LIN {X 0,Y 131.799,Z 543.633,A -85,B 0,C 180,E1 -35494.427,E2 -35494.427} C_VEL
LIN {X 0,Y 126.443,Z 556.276,A -85,B 0,C 180,E1 -35496.559,E2 -35496.559} C_VEL
LIN {X 0,Y 120.613,Z 567.576,A -85,B 0,C 180,E1 -35499.038,E2 -35499.038} C_VEL
LIN {X 0,Y 113.634,Z 578.938,A -85,B 0,C 180,E1 -35502.296,E2 -35502.296} C_VEL
LIN {X 0,Y 106.355,Z 589.12,A -85,B 0,C 180,E1 -35506.25,E2 -35506.25} C_VEL
LIN {X 0,Y 99.674,Z 597.512,A -85,B 0,C 180,E1 -35510.769,E2 -35510.769} C_VEL
LIN {X 0,Y 92.553,Z 605.563,A -85,B 0,C 180,E1 -35516.724,E2 -35516.724} C_VEL
LIN {X 0,Y 86.45,Z 612.057,A -85,B 0,C 180,E1 -35523.537,E2 -35523.537} C_VEL
LIN {X 0,Y 81.061,Z 617.825,A -85,B 0,C 180,E1 -35532.397,E2 -35532.397} C_VEL
LIN {X 0,Y 78.274,Z 621.172,A -85,B 0,C 180,E1 -35539.691,E2 -35539.691} C_VEL
LIN {X 0,Y 76.443,Z 624.336,A -85,B 0,C 180,E1 -35550.001,E2 -35550.001} C_VEL
LIN {X 0,Y 76.754,Z 626.18,A -85,B 0,C 180,E1 -35560.517,E2 -35560.517} C_VEL
LIN {X 0,Y 79.16,Z 626.746,A -85,B 0,C 180,E1 -35570.729,E2 -35570.729} C_VEL
LIN {X 0,Y 83.65,Z 626.018,A -85,B 0,C 180,E1 -35580.161,E2 -35580.161} C_VEL
LIN {X 0,Y 90.169,Z 623.946,A -85,B 0,C 180,E1 -35588.423,E2 -35588.423} C_VEL
LIN {X 0,Y 98.073,Z 620.503,A -85,B 0,C 180,E1 -35595.579,E2 -35595.579} C_VEL
LIN {X 0,Y 107.139,Z 615.57,A -85,B 0,C 180,E1 -35601.678,E2 -35601.678} C_VEL
LIN {X 0,Y 114.562,Z 610.758,A -85,B 0,C 180,E1 -35605.631,E2 -35605.631} C_VEL
LIN {X 0,Y 123.719,Z 603.826,A -85,B 0,C 180,E1 -35609.701,E2 -35609.701} C_VEL
LIN {X 0,Y 127.835,Z 600.345,A -85,B 0,C 180,E1 -35611.246,E2 -35611.246} C_VEL
LIN {X 0,Y 126.024,Z 600.643,A -85,B 0,C 180,E1 -35612.785,E2 -35612.785} C_VEL
LIN {X 0,Y 119.504,Z 603.488,A -85,B 0,C 180,E1 -35615.776,E2 -35615.776} C_VEL
LIN {X 0,Y 106.316,Z 609.311,A -85,B 0,C 180,E1 -35624.719,E2 -35624.719} C_VEL
LIN {X 0,Y 95.376,Z 615.836,A -85,B 0,C 180,E1 -35639.999,E2 -35639.999} C_VEL
LIN {X 0,Y 93.358,Z 619.979,A -85,B 0,C 180,E1 -35653.007,E2 -35653.007} C_VEL
LIN {X 0,Y 99.356,Z 624.746,A -85,B 0,C 180,E1 -35669.569,E2 -35669.569} C_VEL
LIN {X 0,Y 105.626,Z 626.767,A -85,B 0,C 180,E1 -35676.642,E2 -35676.642} C_VEL
LIN {X 0,Y 106.654,Z 627.323,A -85,B 0,C 180,E1 -35677.991,E2 -35677.991} C_VEL
LIN {X 0,Y 98.923,Z 631.915,A -85,B 0,C 180,E1 -35681.971,E2 -35681.971} C_VEL
LIN {X 0,Y 89.878,Z 636.666,A -85,B 0,C 180,E1 -35688.514,E2 -35688.514} C_VEL
LIN {X 0,Y 84.2,Z 639.277,A -85,B 0,C 180,E1 -35694.385,E2 -35694.385} C_VEL
LIN {X 0,Y 78.49,Z 641.629,A -85,B 0,C 180,E1 -35703.499,E2 -35703.499} C_VEL
LIN {X 0,Y 75.481,Z 642.719,A -85,B 0,C 180,E1 -35713.835,E2 -35713.835} C_VEL
LIN {X 0,Y 75.56,Z 642.569,A -85,B 0,C 180,E1 -35724.68,E2 -35724.68} C_VEL
LIN {X 0,Y 78.752,Z 641.176,A -85,B 0,C 180,E1 -35735.102,E2 -35735.102} C_VEL
LIN {X 0,Y 84.849,Z 638.515,A -85,B 0,C 180,E1 -35744.338,E2 -35744.338} C_VEL
LIN {X 0,Y 90.844,Z 635.573,A -85,B 0,C 180,E1 -35750.301,E2 -35750.301} C_VEL
LIN {X 0,Y 97.241,Z 631.893,A -85,B 0,C 180,E1 -35755.423,E2 -35755.423} C_VEL
LIN {X 0,Y 101.803,Z 645.633,A -85,B 0,C 180,E1 -35765.791,E2 -35765.791} C_VEL
LIN {X 0,Y 108.535,Z 655.751,A -85,B 0,C 180,E1 -35773.429,E2 -35773.429} C_VEL
LIN {X 0,Y 109.834,Z 657.283,A -85,B 0,C 180,E1 -35774.547,E2 -35774.547} C_VEL
LIN {X 0,Y 109.87,Z 657.328,A -85,B 0,C 180,E1 -35775.472,E2 -35775.472} C_VEL
LIN {X 0,Y 102.392,Z 646.8,A -85,B 0,C 180,E1 -35783.233,E2 -35783.233} C_VEL
LIN {X 0,Y 98.235,Z 636.568,A -85,B 0,C 180,E1 -35790.858,E2 -35790.858} C_VEL
LIN {X 0,Y 96.502,Z 627.613,A -85,B 0,C 180,E1 -35797.076,E2 -35797.076} C_VEL
LIN {X 0,Y 95.758,Z 622.076,A -85,B 0,C 180,E1 -35800.227,E2 -35800.227} C_VEL
LIN {X 0,Y 93.972,Z 612.024,A -85,B 0,C 180,E1 -35804.325,E2 -35804.325} C_VEL
LIN {X 0,Y 92.54,Z 601.263,A -85,B 0,C 180,E1 -35807.987,E2 -35807.987} C_VEL
LIN {X 0,Y 91.042,Z 586.243,A -85,B 0,C 180,E1 -35812.124,E2 -35812.124} C_VEL
LIN {X 0,Y 89.743,Z 587.101,A -85,B 0,C 180,E1 -35813.278,E2 -35813.278} C_VEL
LIN {X 0,Y 89.136,Z 586.843,A -85,B 0,C 180,E1 -35815.494,E2 -35815.494} C_VEL
LIN {X 0,Y 89.924,Z 585.191,A -85,B 0,C 180,E1 -35817.769,E2 -35817.769} C_VEL
LIN {X 0,Y 89.683,Z 584.831,A -85,B 0,C 180,E1 -35820.001,E2 -35820.001} C_VEL
LIN {X 0,Y 90.085,Z 583.911,A -85,B 0,C 180,E1 -35822.229,E2 -35822.229} C_VEL
LIN {X 0,Y 91.075,Z 582.485,A -85,B 0,C 180,E1 -35824.412,E2 -35824.412} C_VEL
LIN {X 0,Y 92.565,Z 580.529,A -85,B 0,C 180,E1 -35828.706,E2 -35828.706} C_VEL
LIN {X 0,Y 94.154,Z 578.734,A -85,B 0,C 180,E1 -35830.72,E2 -35830.72} C_VEL
LIN {X 0,Y 95.38,Z 577.561,A -85,B 0,C 180,E1 -35832.922,E2 -35832.922} C_VEL
LIN {X 0,Y 96.609,Z 576.576,A -85,B 0,C 180,E1 -35835.156,E2 -35835.156} C_VEL
LIN {X 0,Y 99.926,Z 575.533,A -85,B 0,C 180,E1 -35842.406,E2 -35842.406} C_VEL
LIN {X 0,Y 101.867,Z 574.288,A -85,B 0,C 180,E1 -35844.21,E2 -35844.21} C_VEL
LIN {X 0,Y 102.256,Z 573.98,A -85,B 0,C 180,E1 -35844.45,E2 -35844.45} C_VEL
LIN {X 0,Y 104.721,Z 571.89,A -85,B 0,C 180,E1 -35845.771,E2 -35845.771} C_VEL
LIN {X 0,Y 109.596,Z 568.207,A -85,B 0,C 180,E1 -35848.643,E2 -35848.643} C_VEL
LIN {X 0,Y 115.083,Z 563.519,A -85,B 0,C 180,E1 -35850.952,E2 -35850.952} C_VEL
LIN {X 0,Y 118.67,Z 560.141,A -85,B 0,C 180,E1 -35852.089,E2 -35852.089} C_VEL
LIN {X 0,Y 121.669,Z 557.591,A -85,B 0,C 180,E1 -35853.283,E2 -35853.283} C_VEL
LIN {X 0,Y 122.012,Z 558.369,A -85,B 0,C 180,E1 -35854.086,E2 -35854.086} C_VEL
LIN {X 0,Y 115.629,Z 569.923,A -85,B 0,C 180,E1 -35856.618,E2 -35856.618} C_VEL
LIN {X 0,Y 109.035,Z 580.052,A -85,B 0,C 180,E1 -35859.567,E2 -35859.567} C_VEL
LIN {X 0,Y 101.401,Z 590.161,A -85,B 0,C 180,E1 -35863.506,E2 -35863.506} C_VEL
LIN {X 0,Y 93.404,Z 599.516,A -85,B 0,C 180,E1 -35868.746,E2 -35868.746} C_VEL
LIN {X 0,Y 85.744,Z 607.503,A -85,B 0,C 180,E1 -35875.123,E2 -35875.123} C_VEL
LIN {X 0,Y 80.207,Z 612.967,A -85,B 0,C 180,E1 -35881.295,E2 -35881.295} C_VEL
LIN {X 0,Y 74.377,Z 618.702,A -85,B 0,C 180,E1 -35890.756,E2 -35890.756} C_VEL
LIN {X 0,Y 71.344,Z 622.024,A -85,B 0,C 180,E1 -35898.677,E2 -35898.677} C_VEL
LIN {X 0,Y 69.391,Z 625.153,A -85,B 0,C 180,E1 -35910.001,E2 -35910.001} C_VEL
LIN {X 0,Y 69.794,Z 626.972,A -85,B 0,C 180,E1 -35921.58,E2 -35921.58} C_VEL
LIN {X 0,Y 72.56,Z 627.511,A -85,B 0,C 180,E1 -35932.715,E2 -35932.715} C_VEL
LIN {X 0,Y 77.606,Z 626.752,A -85,B 0,C 180,E1 -35942.79,E2 -35942.79} C_VEL
LIN {X 0,Y 84.715,Z 624.653,A -85,B 0,C 180,E1 -35951.412,E2 -35951.412} C_VEL
LIN {X 0,Y 93.235,Z 621.179,A -85,B 0,C 180,E1 -35958.702,E2 -35958.702} C_VEL
LIN {X 0,Y 102.886,Z 616.213,A -85,B 0,C 180,E1 -35964.783,E2 -35964.783} C_VEL
LIN {X 0,Y 110.708,Z 611.366,A -85,B 0,C 180,E1 -35968.667,E2 -35968.667} C_VEL
LIN {X 0,Y 117.068,Z 606.898,A -85,B 0,C 180,E1 -35971.401,E2 -35971.401} C_VEL
LIN {X 0,Y 117.569,Z 606.1,A -85,B 0,C 180,E1 -35972.501,E2 -35972.501} C_VEL
LIN {X 0,Y 100.067,Z 613.104,A -85,B 0,C 180,E1 -35983.739,E2 -35983.739} C_VEL
LIN {X 0,Y 88.846,Z 619.266,A -85,B 0,C 180,E1 -35999.999,E2 -35999.999} C_VEL
LIN {X 0,Y 87.017,Z 623.184,A -85,B 0,C 180,E1 -36013.973,E2 -36013.973} C_VEL
LIN {X 0,Y 93.708,Z 627.77,A -85,B 0,C 180,E1 -36031.548,E2 -36031.548} C_VEL
LIN {X 0,Y 96.799,Z 628.787,A -85,B 0,C 180,E1 -36035.371,E2 -36035.371} C_VEL
LIN {X 0,Y 96.943,Z 629.812,A -85,B 0,C 180,E1 -36037.363,E2 -36037.363} C_VEL
LIN {X 0,Y 86.962,Z 634.909,A -85,B 0,C 180,E1 -36043.537,E2 -36043.537} C_VEL
LIN {X 0,Y 78.535,Z 638.568,A -85,B 0,C 180,E1 -36051.366,E2 -36051.366} C_VEL
LIN {X 0,Y 72.174,Z 640.888,A -85,B 0,C 180,E1 -36060.97,E2 -36060.97} C_VEL
LIN {X 0,Y 68.647,Z 641.949,A -85,B 0,C 180,E1 -36072.174,E2 -36072.174} C_VEL
LIN {X 0,Y 68.404,Z 641.766,A -85,B 0,C 180,E1 -36084.122,E2 -36084.122} C_VEL
LIN {X 0,Y 71.571,Z 640.342,A -85,B 0,C 180,E1 -36095.615,E2 -36095.615} C_VEL
LIN {X 0,Y 77.861,Z 637.643,A -85,B 0,C 180,E1 -36105.656,E2 -36105.656} C_VEL
LIN {X 0,Y 84.186,Z 634.651,A -85,B 0,C 180,E1 -36112.056,E2 -36112.056} C_VEL
LIN {X 0,Y 92.43,Z 629.904,A -85,B 0,C 180,E1 -36118.593,E2 -36118.593} C_VEL
LIN {X 0,Y 93.542,Z 629.553,A -85,B 0,C 180,E1 -36119.188,E2 -36119.188} C_VEL
LIN {X 0,Y 97.855,Z 641.235,A -85,B 0,C 180,E1 -36128.06,E2 -36128.06} C_VEL
LIN {X 0,Y 102.156,Z 648.086,A -85,B 0,C 180,E1 -36133.287,E2 -36133.287} C_VEL
LIN {X 0,Y 103.341,Z 649.651,A -85,B 0,C 180,E1 -36135.582,E2 -36135.582} C_VEL
LIN {X 0,Y 96.168,Z 637.856,A -85,B 0,C 180,E1 -36144.362,E2 -36144.362} C_VEL
LIN {X 0,Y 92.965,Z 627.766,A -85,B 0,C 180,E1 -36151.851,E2 -36151.851} C_VEL
LIN {X 0,Y 91.738,Z 620.852,A -85,B 0,C 180,E1 -36156.38,E2 -36156.38} C_VEL
LIN {X 0,Y 90.34,Z 613.827,A -85,B 0,C 180,E1 -36159.581,E2 -36159.581} C_VEL
LIN {X 0,Y 88.299,Z 602.174,A -85,B 0,C 180,E1 -36163.882,E2 -36163.882} C_VEL
LIN {X 0,Y 86.997,Z 593.297,A -85,B 0,C 180,E1 -36166.612,E2 -36166.612} C_VEL
LIN {X 0,Y 86.234,Z 593.75,A -85,B 0,C 180,E1 -36167.084,E2 -36167.084} C_VEL
LIN {X 0,Y 84.539,Z 593.631,A -85,B 0,C 180,E1 -36170.463,E2 -36170.463} C_VEL
LIN {X 0,Y 84.831,Z 592.553,A -85,B 0,C 180,E1 -36172.232,E2 -36172.232} C_VEL
LIN {X 0,Y 84.181,Z 591.51,A -85,B 0,C 180,E1 -36176.83,E2 -36176.83} C_VEL
LIN {X 0,Y 84.828,Z 590.014,A -85,B 0,C 180,E1 -36180.001,E2 -36180.001} C_VEL
LIN {X 0,Y 85.83,Z 588.22,A -85,B 0,C 180,E1 -36184.682,E2 -36184.682} C_VEL
LIN {X 0,Y 88.893,Z 584.872,A -85,B 0,C 180,E1 -36191.362,E2 -36191.362} C_VEL
LIN {X 0,Y 90.544,Z 583.299,A -85,B 0,C 180,E1 -36193.421,E2 -36193.421} C_VEL
LIN {X 0,Y 93.583,Z 580.842,A -85,B 0,C 180,E1 -36197.422,E2 -36197.422} C_VEL
LIN {X 0,Y 97.615,Z 577.561,A -85,B 0,C 180,E1 -36201.026,E2 -36201.026} C_VEL
LIN {X 0,Y 99.606,Z 576.094,A -85,B 0,C 180,E1 -36202.755,E2 -36202.755} C_VEL
LIN {X 0,Y 102.256,Z 573.98,A -85,B 0,C 180,E1 -36204.45,E2 -36204.45} C_VEL
LIN {X 0,Y 103.756,Z 573.102,A -85,B 0,C 180,E1 -36205.758,E2 -36205.758} C_VEL
LIN {X 0,Y 104.922,Z 573.264,A -85,B 0,C 180,E1 -36207.784,E2 -36207.784} C_VEL
LIN {X 0,Y 105.476,Z 574.59,A -85,B 0,C 180,E1 -36210.177,E2 -36210.177} C_VEL
LIN {X 0,Y 105.226,Z 577.34,A -85,B 0,C 180,E1 -36212.996,E2 -36212.996} C_VEL
LIN {X 0,Y 103.788,Z 581.57,A -85,B 0,C 180,E1 -36216.102,E2 -36216.102} C_VEL
LIN {X 0,Y 101.776,Z 584.935,A -85,B 0,C 180,E1 -36217.892,E2 -36217.892} C_VEL
LIN {X 0,Y 101.257,Z 585.634,A -85,B 0,C 180,E1 -36218.177,E2 -36218.177} C_VEL
LIN {X 0,Y 94.139,Z 594.118,A -85,B 0,C 180,E1 -36221.923,E2 -36221.923} C_VEL
LIN {X 0,Y 85.695,Z 603.123,A -85,B 0,C 180,E1 -36227.599,E2 -36227.599} C_VEL
LIN {X 0,Y 77.958,Z 610.402,A -85,B 0,C 180,E1 -36234.267,E2 -36234.267} C_VEL
LIN {X 0,Y 70.694,Z 616.928,A -85,B 0,C 180,E1 -36243.522,E2 -36243.522} C_VEL
LIN {X 0,Y 65.881,Z 621.364,A -85,B 0,C 180,E1 -36253.12,E2 -36253.12} C_VEL
LIN {X 0,Y 63.053,Z 624.59,A -85,B 0,C 180,E1 -36263.623,E2 -36263.623} C_VEL
LIN {X 0,Y 62.226,Z 627.032,A -85,B 0,C 180,E1 -36276.464,E2 -36276.464} C_VEL
LIN {X 0,Y 64.178,Z 628.176,A -85,B 0,C 180,E1 -36289.114,E2 -36289.114} C_VEL
LIN {X 0,Y 68.595,Z 628.048,A -85,B 0,C 180,E1 -36300.703,E2 -36300.703} C_VEL
LIN {X 0,Y 75.46,Z 626.586,A -85,B 0,C 180,E1 -36310.525,E2 -36310.525} C_VEL
LIN {X 0,Y 83.964,Z 623.785,A -85,B 0,C 180,E1 -36318.661,E2 -36318.661} C_VEL
LIN {X 0,Y 93.723,Z 619.55,A -85,B 0,C 180,E1 -36325.296,E2 -36325.296} C_VEL
LIN {X 0,Y 104.376,Z 613.743,A -85,B 0,C 180,E1 -36330.741,E2 -36330.741} C_VEL
LIN {X 0,Y 106.313,Z 612.521,A -85,B 0,C 180,E1 -36331.557,E2 -36331.557} C_VEL
LIN {X 0,Y 107.708,Z 611.402,A -85,B 0,C 180,E1 -36332.92,E2 -36332.92} C_VEL
LIN {X 0,Y 93.695,Z 616.547,A -85,B 0,C 180,E1 -36342.599,E2 -36342.599} C_VEL
LIN {X 0,Y 82.168,Z 622.361,A -85,B 0,C 180,E1 -36359.999,E2 -36359.999} C_VEL
LIN {X 0,Y 80.537,Z 626.085,A -85,B 0,C 180,E1 -36375.123,E2 -36375.123} C_VEL
LIN {X 0,Y 88.795,Z 630.692,A -85,B 0,C 180,E1 -36394.745,E2 -36394.745} C_VEL
LIN {X 0,Y 87.348,Z 631.883,A -85,B 0,C 180,E1 -36396.686,E2 -36396.686} C_VEL
LIN {X 0,Y 77.449,Z 636.215,A -85,B 0,C 180,E1 -36403.653,E2 -36403.653} C_VEL
LIN {X 0,Y 69.302,Z 639.169,A -85,B 0,C 180,E1 -36412.667,E2 -36412.667} C_VEL
LIN {X 0,Y 63.543,Z 640.819,A -85,B 0,C 180,E1 -36423.836,E2 -36423.836} C_VEL
LIN {X 0,Y 61.12,Z 641.229,A -85,B 0,C 180,E1 -36436.749,E2 -36436.749} C_VEL
LIN {X 0,Y 62.386,Z 640.393,A -85,B 0,C 180,E1 -36449.999,E2 -36449.999} C_VEL
LIN {X 0,Y 67.284,Z 638.301,A -85,B 0,C 180,E1 -36462.016,E2 -36462.016} C_VEL
LIN {X 0,Y 75.159,Z 634.878,A -85,B 0,C 180,E1 -36471.886,E2 -36471.886} C_VEL
LIN {X 0,Y 82.141,Z 631.313,A -85,B 0,C 180,E1 -36477.969,E2 -36477.969} C_VEL
LIN {X 0,Y 89.66,Z 627.053,A -85,B 0,C 180,E1 -36482.817,E2 -36482.817} C_VEL
LIN {X 0,Y 90.096,Z 626.893,A -85,B 0,C 180,E1 -36482.97,E2 -36482.97} C_VEL
LIN {X 0,Y 94.992,Z 638.061,A -85,B 0,C 180,E1 -36491.577,E2 -36491.577} C_VEL
LIN {X 0,Y 96.614,Z 640.612,A -85,B 0,C 180,E1 -36493.533,E2 -36493.533} C_VEL
LIN {X 0,Y 97.62,Z 642.119,A -85,B 0,C 180,E1 -36495.311,E2 -36495.311} C_VEL
LIN {X 0,Y 90.924,Z 629.599,A -85,B 0,C 180,E1 -36504.705,E2 -36504.705} C_VEL
LIN {X 0,Y 88.298,Z 620.143,A -85,B 0,C 180,E1 -36511.579,E2 -36511.579} C_VEL
LIN {X 0,Y 87.572,Z 616.386,A -85,B 0,C 180,E1 -36513.903,E2 -36513.903} C_VEL
LIN {X 0,Y 85.261,Z 606.269,A -85,B 0,C 180,E1 -36518.146,E2 -36518.146} C_VEL
LIN {X 0,Y 83.987,Z 599.658,A -85,B 0,C 180,E1 -36520.514,E2 -36520.514} C_VEL
LIN {X 0,Y 80.764,Z 599.708,A -85,B 0,C 180,E1 -36524.92,E2 -36524.92} C_VEL
LIN {X 0,Y 79.439,Z 598.471,A -85,B 0,C 180,E1 -36529.844,E2 -36529.844} C_VEL
LIN {X 0,Y 79.446,Z 595.225,A -85,B 0,C 180,E1 -36540.001,E2 -36540.001} C_VEL
LIN {X 0,Y 83.733,Z 590.303,A -85,B 0,C 180,E1 -36552.073,E2 -36552.073} C_VEL
LIN {X 0,Y 90.536,Z 585.126,A -85,B 0,C 180,E1 -36560.375,E2 -36560.375} C_VEL
LIN {X 0,Y 95.546,Z 581.56,A -85,B 0,C 180,E1 -36564.439,E2 -36564.439} C_VEL
LIN {X 0,Y 97.123,Z 580.531,A -85,B 0,C 180,E1 -36565.641,E2 -36565.641} C_VEL
LIN {X 0,Y 102.573,Z 576.509,A -85,B 0,C 180,E1 -36568.557,E2 -36568.557} C_VEL
LIN {X 0,Y 107.839,Z 572.89,A -85,B 0,C 180,E1 -36571.308,E2 -36571.308} C_VEL
LIN {X 0,Y 111.957,Z 569.78,A -85,B 0,C 180,E1 -36572.959,E2 -36572.959} C_VEL
LIN {X 0,Y 111.584,Z 571.099,A -85,B 0,C 180,E1 -36573.723,E2 -36573.723} C_VEL
LIN {X 0,Y 104.707,Z 581.162,A -85,B 0,C 180,E1 -36576.607,E2 -36576.607} C_VEL
LIN {X 0,Y 101.257,Z 585.634,A -85,B 0,C 180,E1 -36578.177,E2 -36578.177} C_VEL
LIN {X 0,Y 97.678,Z 589.729,A -85,B 0,C 180,E1 -36579.505,E2 -36579.505} C_VEL
LIN {X 0,Y 90.585,Z 596.138,A -85,B 0,C 180,E1 -36581.108,E2 -36581.108} C_VEL
LIN {X 0,Y 83.198,Z 602.029,A -85,B 0,C 180,E1 -36583.121,E2 -36583.121} C_VEL
LIN {X 0,Y 79.264,Z 605.314,A -85,B 0,C 180,E1 -36585.205,E2 -36585.205} C_VEL
LIN {X 0,Y 72.354,Z 611.331,A -85,B 0,C 180,E1 -36591.006,E2 -36591.006} C_VEL
LIN {X 0,Y 64.465,Z 617.822,A -85,B 0,C 180,E1 -36600.729,E2 -36600.729} C_VEL
LIN {X 0,Y 59.602,Z 621.871,A -85,B 0,C 180,E1 -36610.083,E2 -36610.083} C_VEL
LIN {X 0,Y 56.034,Z 625.423,A -85,B 0,C 180,E1 -36622.82,E2 -36622.82} C_VEL
LIN {X 0,Y 55.211,Z 627.836,A -85,B 0,C 180,E1 -36637.29,E2 -36637.29} C_VEL
LIN {X 0,Y 57.527,Z 628.954,A -85,B 0,C 180,E1 -36651.426,E2 -36651.426} C_VEL
LIN {X 0,Y 62.595,Z 628.798,A -85,B 0,C 180,E1 -36664.023,E2 -36664.023} C_VEL
LIN {X 0,Y 70.224,Z 627.305,A -85,B 0,C 180,E1 -36674.285,E2 -36674.285} C_VEL
LIN {X 0,Y 79.452,Z 624.477,A -85,B 0,C 180,E1 -36682.51,E2 -36682.51} C_VEL
LIN {X 0,Y 89.869,Z 620.21,A -85,B 0,C 180,E1 -36689.021,E2 -36689.021} C_VEL
LIN {X 0,Y 95.396,Z 617.5,A -85,B 0,C 180,E1 -36691.777,E2 -36691.777} C_VEL
LIN {X 0,Y 97.601,Z 616.136,A -85,B 0,C 180,E1 -36693.486,E2 -36693.486} C_VEL
LIN {X 0,Y 87.216,Z 619.648,A -85,B 0,C 180,E1 -36701.26,E2 -36701.26} C_VEL
LIN {X 0,Y 75.347,Z 625.119,A -85,B 0,C 180,E1 -36719.999,E2 -36719.999} C_VEL
LIN {X 0,Y 74.009,Z 628.648,A -85,B 0,C 180,E1 -36736.493,E2 -36736.493} C_VEL
LIN {X 0,Y 80.169,Z 632.1,A -85,B 0,C 180,E1 -36753.089,E2 -36753.089} C_VEL
LIN {X 0,Y 79.538,Z 632.862,A -85,B 0,C 180,E1 -36754.903,E2 -36754.903} C_VEL
LIN {X 0,Y 72.721,Z 635.521,A -85,B 0,C 180,E1 -36759.595,E2 -36759.595} C_VEL
LIN {X 0,Y 63.778,Z 638.443,A -85,B 0,C 180,E1 -36768.778,E2 -36768.778} C_VEL
LIN {X 0,Y 57.218,Z 640.064,A -85,B 0,C 180,E1 -36780.68,E2 -36780.68} C_VEL
LIN {X 0,Y 54.163,Z 640.441,A -85,B 0,C 180,E1 -36795.009,E2 -36795.009} C_VEL
LIN {X 0,Y 55.211,Z 639.573,A -85,B 0,C 180,E1 -36809.999,E2 -36809.999} C_VEL
LIN {X 0,Y 60.24,Z 637.441,A -85,B 0,C 180,E1 -36823.446,E2 -36823.446} C_VEL
LIN {X 0,Y 68.508,Z 633.983,A -85,B 0,C 180,E1 -36834.139,E2 -36834.139} C_VEL
LIN {X 0,Y 75.896,Z 630.411,A -85,B 0,C 180,E1 -36840.503,E2 -36840.503} C_VEL
LIN {X 0,Y 83.983,Z 625.892,A -85,B 0,C 180,E1 -36845.719,E2 -36845.719} C_VEL
LIN {X 0,Y 87.273,Z 624.32,A -85,B 0,C 180,E1 -36847.188,E2 -36847.188} C_VEL
LIN {X 0,Y 91.302,Z 632.685,A -85,B 0,C 180,E1 -36853.665,E2 -36853.665} C_VEL
LIN {X 0,Y 91.964,Z 633.773,A -85,B 0,C 180,E1 -36855.427,E2 -36855.427} C_VEL
LIN {X 0,Y 85.947,Z 620.765,A -85,B 0,C 180,E1 -36865.217,E2 -36865.217} C_VEL
LIN {X 0,Y 84.137,Z 613.79,A -85,B 0,C 180,E1 -36870.034,E2 -36870.034} C_VEL
LIN {X 0,Y 82.033,Z 605.772,A -85,B 0,C 180,E1 -36873.582,E2 -36873.582} C_VEL
LIN {X 0,Y 80.584,Z 606.256,A -85,B 0,C 180,E1 -36874.241,E2 -36874.241} C_VEL
LIN {X 0,Y 74.079,Z 603.105,A -85,B 0,C 180,E1 -36889.101,E2 -36889.101} C_VEL
LIN {X 0,Y 73.996,Z 600.009,A -85,B 0,C 180,E1 -36900.001,E2 -36900.001} C_VEL
LIN {X 0,Y 79.842,Z 594.304,A -85,B 0,C 180,E1 -36915.202,E2 -36915.202} C_VEL
LIN {X 0,Y 87.572,Z 589.219,A -85,B 0,C 180,E1 -36923.575,E2 -36923.575} C_VEL
LIN {X 0,Y 92.333,Z 586.185,A -85,B 0,C 180,E1 -36927.077,E2 -36927.077} C_VEL
LIN {X 0,Y 96.923,Z 583.369,A -85,B 0,C 180,E1 -36929.864,E2 -36929.864} C_VEL
LIN {X 0,Y 101.719,Z 580.162,A -85,B 0,C 180,E1 -36932.105,E2 -36932.105} C_VEL
LIN {X 0,Y 101.525,Z 581.123,A -85,B 0,C 180,E1 -36933.039,E2 -36933.039} C_VEL
LIN {X 0,Y 93.671,Z 590.686,A -85,B 0,C 180,E1 -36936.501,E2 -36936.501} C_VEL
LIN {X 0,Y 85.799,Z 599.07,A -85,B 0,C 180,E1 -36940.778,E2 -36940.778} C_VEL
LIN {X 0,Y 79.264,Z 605.314,A -85,B 0,C 180,E1 -36945.205,E2 -36945.205} C_VEL
LIN {X 0,Y 75.347,Z 608.457,A -85,B 0,C 180,E1 -36947.551,E2 -36947.551} C_VEL
LIN {X 0,Y 67.823,Z 613.26,A -85,B 0,C 180,E1 -36951.038,E2 -36951.038} C_VEL
LIN {X 0,Y 60.449,Z 617.565,A -85,B 0,C 180,E1 -36955.563,E2 -36955.563} C_VEL
LIN {X 0,Y 56.976,Z 619.797,A -85,B 0,C 180,E1 -36959.645,E2 -36959.645} C_VEL
LIN {X 0,Y 51.948,Z 623.574,A -85,B 0,C 180,E1 -36970.302,E2 -36970.302} C_VEL
LIN {X 0,Y 49.053,Z 626.254,A -85,B 0,C 180,E1 -36981.792,E2 -36981.792} C_VEL
LIN {X 0,Y 48.222,Z 628.639,A -85,B 0,C 180,E1 -36998.353,E2 -36998.353} C_VEL
LIN {X 0,Y 50.986,Z 629.732,A -85,B 0,C 180,E1 -37014.341,E2 -37014.341} C_VEL
LIN {X 0,Y 56.85,Z 629.547,A -85,B 0,C 180,E1 -37028.029,E2 -37028.029} C_VEL
LIN {X 0,Y 65.34,Z 628.025,A -85,B 0,C 180,E1 -37038.627,E2 -37038.627} C_VEL
LIN {X 0,Y 75.339,Z 625.168,A -85,B 0,C 180,E1 -37046.8,E2 -37046.8} C_VEL
LIN {X 0,Y 86.422,Z 620.871,A -85,B 0,C 180,E1 -37053.07,E2 -37053.07} C_VEL
LIN {X 0,Y 87.375,Z 620.361,A -85,B 0,C 180,E1 -37054.139,E2 -37054.139} C_VEL
LIN {X 0,Y 73.249,Z 625.05,A -85,B 0,C 180,E1 -37068.973,E2 -37068.973} C_VEL
LIN {X 0,Y 67.193,Z 628.695,A -85,B 0,C 180,E1 -37085.982,E2 -37085.982} C_VEL
LIN {X 0,Y 70.909,Z 632.954,A -85,B 0,C 180,E1 -37109.596,E2 -37109.596} C_VEL
LIN {X 0,Y 71.629,Z 633.237,A -85,B 0,C 180,E1 -37111.101,E2 -37111.101} C_VEL
LIN {X 0,Y 71.567,Z 633.744,A -85,B 0,C 180,E1 -37112.899,E2 -37112.899} C_VEL
LIN {X 0,Y 63.285,Z 636.44,A -85,B 0,C 180,E1 -37119.214,E2 -37119.214} C_VEL
LIN {X 0,Y 54.499,Z 638.673,A -85,B 0,C 180,E1 -37130.011,E2 -37130.011} C_VEL
LIN {X 0,Y 48.672,Z 639.636,A -85,B 0,C 180,E1 -37144.421,E2 -37144.421} C_VEL
LIN {X 0,Y 47.065,Z 639.356,A -85,B 0,C 180,E1 -37161.44,E2 -37161.44} C_VEL
LIN {X 0,Y 50.108,Z 637.821,A -85,B 0,C 180,E1 -37178.034,E2 -37178.034} C_VEL
LIN {X 0,Y 57.272,Z 635.005,A -85,B 0,C 180,E1 -37191.524,E2 -37191.524} C_VEL
LIN {X 0,Y 67.135,Z 630.79,A -85,B 0,C 180,E1 -37201.444,E2 -37201.444} C_VEL
LIN {X 0,Y 78.283,Z 624.955,A -85,B 0,C 180,E1 -37208.779,E2 -37208.779} C_VEL
LIN {X 0,Y 84.685,Z 621.46,A -85,B 0,C 180,E1 -37211.429,E2 -37211.429} C_VEL
LIN {X 0,Y 85.136,Z 621.898,A -85,B 0,C 180,E1 -37211.869,E2 -37211.869} C_VEL
LIN {X 0,Y 86.276,Z 624.167,A -85,B 0,C 180,E1 -37213.639,E2 -37213.639} C_VEL
LIN {X 0,Y 86.668,Z 624.938,A -85,B 0,C 180,E1 -37215.602,E2 -37215.602} C_VEL
LIN {X 0,Y 82.219,Z 614.608,A -85,B 0,C 180,E1 -37223.393,E2 -37223.393} C_VEL
LIN {X 0,Y 81.48,Z 612.205,A -85,B 0,C 180,E1 -37225.097,E2 -37225.097} C_VEL
LIN {X 0,Y 80.459,Z 612.39,A -85,B 0,C 180,E1 -37225.539,E2 -37225.539} C_VEL
LIN {X 0,Y 78.242,Z 612.139,A -85,B 0,C 180,E1 -37227.513,E2 -37227.513} C_VEL
LIN {X 0,Y 75.523,Z 610.526,A -85,B 0,C 180,E1 -37232.373,E2 -37232.373} C_VEL
LIN {X 0,Y 68.524,Z 607.469,A -85,B 0,C 180,E1 -37248.205,E2 -37248.205} C_VEL
LIN {X 0,Y 69.545,Z 602.859,A -85,B 0,C 180,E1 -37265.782,E2 -37265.782} C_VEL
LIN {X 0,Y 75.785,Z 598.255,A -85,B 0,C 180,E1 -37278.325,E2 -37278.325} C_VEL
LIN {X 0,Y 84.733,Z 593.113,A -85,B 0,C 180,E1 -37287.044,E2 -37287.044} C_VEL
LIN {X 0,Y 88.606,Z 590.872,A -85,B 0,C 180,E1 -37289.592,E2 -37289.592} C_VEL
LIN {X 0,Y 91.099,Z 590.143,A -85,B 0,C 180,E1 -37292.246,E2 -37292.246} C_VEL
LIN {X 0,Y 82.333,Z 599.15,A -85,B 0,C 180,E1 -37296.491,E2 -37296.491} C_VEL
LIN {X 0,Y 73.267,Z 607.265,A -85,B 0,C 180,E1 -37302.192,E2 -37302.192} C_VEL
LIN {X 0,Y 64.713,Z 614.042,A -85,B 0,C 180,E1 -37309.502,E2 -37309.502} C_VEL
LIN {X 0,Y 56.976,Z 619.797,A -85,B 0,C 180,E1 -37319.645,E2 -37319.645} C_VEL
LIN {X 0,Y 53.773,Z 621.918,A -85,B 0,C 180,E1 -37324.288,E2 -37324.288} C_VEL
LIN {X 0,Y 47.623,Z 625.027,A -85,B 0,C 180,E1 -37332.362,E2 -37332.362} C_VEL
LIN {X 0,Y 43.277,Z 627.025,A -85,B 0,C 180,E1 -37340.408,E2 -37340.408} C_VEL
LIN {X 0,Y 41.342,Z 628.178,A -85,B 0,C 180,E1 -37347.846,E2 -37347.846} C_VEL
LIN {X 0,Y 41.102,Z 628.484,A -85,B 0,C 180,E1 -37350.541,E2 -37350.541} C_VEL
LIN {X 0,Y 42.437,Z 630.136,A -85,B 0,C 180,E1 -37369.277,E2 -37369.277} C_VEL
LIN {X 0,Y 47.666,Z 630.565,A -85,B 0,C 180,E1 -37386.002,E2 -37386.002} C_VEL
LIN {X 0,Y 55.95,Z 629.684,A -85,B 0,C 180,E1 -37398.692,E2 -37398.692} C_VEL
LIN {X 0,Y 66.762,Z 627.319,A -85,B 0,C 180,E1 -37408.358,E2 -37408.358} C_VEL
LIN {X 0,Y 74.271,Z 625.016,A -85,B 0,C 180,E1 -37413.01,E2 -37413.01} C_VEL
LIN {X 0,Y 76.714,Z 624.086,A -85,B 0,C 180,E1 -37415.382,E2 -37415.382} C_VEL
LIN {X 0,Y 63.421,Z 628.51,A -85,B 0,C 180,E1 -37433.73,E2 -37433.73} C_VEL
LIN {X 0,Y 60.043,Z 631.757,A -85,B 0,C 180,E1 -37453.491,E2 -37453.491} C_VEL
LIN {X 0,Y 63.195,Z 634.095,A -85,B 0,C 180,E1 -37468.614,E2 -37468.614} C_VEL
LIN {X 0,Y 62.926,Z 634.637,A -85,B 0,C 180,E1 -37470.949,E2 -37470.949} C_VEL
LIN {X 0,Y 53.89,Z 636.994,A -85,B 0,C 180,E1 -37478.75,E2 -37478.75} C_VEL
LIN {X 0,Y 45.321,Z 638.549,A -85,B 0,C 180,E1 -37491.812,E2 -37491.812} C_VEL
LIN {X 0,Y 40.486,Z 638.855,A -85,B 0,C 180,E1 -37509.754,E2 -37509.754} C_VEL
LIN {X 0,Y 40.844,Z 637.918,A -85,B 0,C 180,E1 -37529.998,E2 -37529.998} C_VEL
LIN {X 0,Y 46.311,Z 635.71,A -85,B 0,C 180,E1 -37547.606,E2 -37547.606} C_VEL
LIN {X 0,Y 55.619,Z 632.188,A -85,B 0,C 180,E1 -37560.247,E2 -37560.247} C_VEL
LIN {X 0,Y 66.859,Z 627.163,A -85,B 0,C 180,E1 -37568.945,E2 -37568.945} C_VEL
LIN {X 0,Y 76.052,Z 622.316,A -85,B 0,C 180,E1 -37573.693,E2 -37573.693} C_VEL
LIN {X 0,Y 79.426,Z 620.319,A -85,B 0,C 180,E1 -37575.131,E2 -37575.131} C_VEL
LIN {X 0,Y 76.353,Z 618.025,A -85,B 0,C 180,E1 -37580.048,E2 -37580.048} C_VEL
LIN {X 0,Y 73.351,Z 616.068,A -85,B 0,C 180,E1 -37585.045,E2 -37585.045} C_VEL
LIN {X 0,Y 70.24,Z 614.627,A -85,B 0,C 180,E1 -37590.094,E2 -37590.094} C_VEL
LIN {X 0,Y 62.811,Z 611.538,A -85,B 0,C 180,E1 -37607.114,E2 -37607.114} C_VEL
LIN {X 0,Y 63.707,Z 607.166,A -85,B 0,C 180,E1 -37626.314,E2 -37626.314} C_VEL
LIN {X 0,Y 70.891,Z 602.487,A -85,B 0,C 180,E1 -37640.728,E2 -37640.728} C_VEL
LIN {X 0,Y 80.859,Z 597.415,A -85,B 0,C 180,E1 -37649.975,E2 -37649.975} C_VEL
LIN {X 0,Y 81.578,Z 597.208,A -85,B 0,C 180,E1 -37650.84,E2 -37650.84} C_VEL
LIN {X 0,Y 71.524,Z 606.028,A -85,B 0,C 180,E1 -37656.107,E2 -37656.107} C_VEL
LIN {X 0,Y 62.043,Z 613.187,A -85,B 0,C 180,E1 -37662.793,E2 -37662.793} C_VEL
LIN {X 0,Y 52.631,Z 619.609,A -85,B 0,C 180,E1 -37673.211,E2 -37673.211} C_VEL
LIN {X 0,Y 45.375,Z 624.436,A -85,B 0,C 180,E1 -37687.301,E2 -37687.301} C_VEL
LIN {X 0,Y 42.084,Z 627.086,A -85,B 0,C 180,E1 -37700.421,E2 -37700.421} C_VEL
LIN {X 0,Y 41.102,Z 628.484,A -85,B 0,C 180,E1 -37710.541,E2 -37710.541} C_VEL
LIN {X 0,Y 40.48,Z 629.429,A -85,B 0,C 180,E1 -37718.715,E2 -37718.715} C_VEL
LIN {X 0,Y 39.441,Z 630.63,A -85,B 0,C 180,E1 -37732.786,E2 -37732.786} C_VEL
LIN {X 0,Y 40.146,Z 631.218,A -85,B 0,C 180,E1 -37744.197,E2 -37744.197} C_VEL
LIN {X 0,Y 42.322,Z 631.318,A -85,B 0,C 180,E1 -37751.869,E2 -37751.869} C_VEL
LIN {X 0,Y 43.416,Z 631.241,A -85,B 0,C 180,E1 -37754.068,E2 -37754.068} C_VEL
LIN {X 0,Y 51.547,Z 630.419,A -85,B 0,C 180,E1 -37764.621,E2 -37764.621} C_VEL
LIN {X 0,Y 62.81,Z 628.147,A -85,B 0,C 180,E1 -37773.506,E2 -37773.506} C_VEL
LIN {X 0,Y 64.119,Z 627.832,A -85,B 0,C 180,E1 -37774.317,E2 -37774.317} C_VEL
LIN {X 0,Y 66.358,Z 627.169,A -85,B 0,C 180,E1 -37776.789,E2 -37776.789} C_VEL
LIN {X 0,Y 54.261,Z 631.349,A -85,B 0,C 180,E1 -37799.998,E2 -37799.998} C_VEL
LIN {X 0,Y 55.403,Z 635.022,A -85,B 0,C 180,E1 -37827.747,E2 -37827.747} C_VEL
LIN {X 0,Y 44.557,Z 637.189,A -85,B 0,C 180,E1 -37838.184,E2 -37838.184} C_VEL
LIN {X 0,Y 36.315,Z 638.079,A -85,B 0,C 180,E1 -37854.643,E2 -37854.643} C_VEL
LIN {X 0,Y 32.948,Z 637.729,A -85,B 0,C 180,E1 -37877.724,E2 -37877.724} C_VEL
LIN {X 0,Y 35.887,Z 636.123,A -85,B 0,C 180,E1 -37901.253,E2 -37901.253} C_VEL
LIN {X 0,Y 44.146,Z 633.242,A -85,B 0,C 180,E1 -37918.423,E2 -37918.423} C_VEL
LIN {X 0,Y 55.34,Z 628.967,A -85,B 0,C 180,E1 -37929.259,E2 -37929.259} C_VEL
LIN {X 0,Y 64.54,Z 624.739,A -85,B 0,C 180,E1 -37934.864,E2 -37934.864} C_VEL
LIN {X 0,Y 70.58,Z 621.595,A -85,B 0,C 180,E1 -37937.546,E2 -37937.546} C_VEL
LIN {X 0,Y 68.188,Z 619.921,A -85,B 0,C 180,E1 -37941.953,E2 -37941.953} C_VEL
LIN {X 0,Y 64.981,Z 618.393,A -85,B 0,C 180,E1 -37947.389,E2 -37947.389} C_VEL
LIN {X 0,Y 56.952,Z 615.316,A -85,B 0,C 180,E1 -37965.762,E2 -37965.762} C_VEL
LIN {X 0,Y 56.401,Z 612.672,A -85,B 0,C 180,E1 -37980.002,E2 -37980.002} C_VEL
LIN {X 0,Y 59.957,Z 609.565,A -85,B 0,C 180,E1 -37993.514,E2 -37993.514} C_VEL
LIN {X 0,Y 66.984,Z 605.951,A -85,B 0,C 180,E1 -38004.728,E2 -38004.728} C_VEL
LIN {X 0,Y 71.698,Z 603.774,A -85,B 0,C 180,E1 -38009.242,E2 -38009.242} C_VEL
LIN {X 0,Y 63.192,Z 610.248,A -85,B 0,C 180,E1 -38013.766,E2 -38013.766} C_VEL
LIN {X 0,Y 54.776,Z 615.898,A -85,B 0,C 180,E1 -38019.895,E2 -38019.895} C_VEL
LIN {X 0,Y 47.191,Z 620.501,A -85,B 0,C 180,E1 -38028.095,E2 -38028.095} C_VEL
LIN {X 0,Y 38.965,Z 625.298,A -85,B 0,C 180,E1 -38043.296,E2 -38043.296} C_VEL
LIN {X 0,Y 35.133,Z 627.92,A -85,B 0,C 180,E1 -38058.502,E2 -38058.502} C_VEL
LIN {X 0,Y 34.276,Z 630.25,A -85,B 0,C 180,E1 -38081.794,E2 -38081.794} C_VEL
LIN {X 0,Y 38.523,Z 631.287,A -85,B 0,C 180,E1 -38103.059,E2 -38103.059} C_VEL
LIN {X 0,Y 43.416,Z 631.241,A -85,B 0,C 180,E1 -38114.068,E2 -38114.068} C_VEL
LIN {X 0,Y 45.449,Z 631.175,A -85,B 0,C 180,E1 -38118.458,E2 -38118.458} C_VEL
LIN {X 0,Y 48.057,Z 630.99,A -85,B 0,C 180,E1 -38126.008,E2 -38126.008} C_VEL
LIN {X 0,Y 52.025,Z 630.493,A -85,B 0,C 180,E1 -38134.086,E2 -38134.086} C_VEL
LIN {X 0,Y 53.916,Z 630.144,A -85,B 0,C 180,E1 -38136.11,E2 -38136.11} C_VEL
LIN {X 0,Y 56.413,Z 629.659,A -85,B 0,C 180,E1 -38138.128,E2 -38138.128} C_VEL
LIN {X 0,Y 47.111,Z 632.728,A -85,B 0,C 180,E1 -38159.998,E2 -38159.998} C_VEL
LIN {X 0,Y 46.341,Z 634.636,A -85,B 0,C 180,E1 -38177.593,E2 -38177.593} C_VEL
LIN {X 0,Y 46.334,Z 635.534,A -85,B 0,C 180,E1 -38184.897,E2 -38184.897} C_VEL
LIN {X 0,Y 35.241,Z 637.021,A -85,B 0,C 180,E1 -38197.337,E2 -38197.337} C_VEL
LIN {X 0,Y 27.502,Z 637.257,A -85,B 0,C 180,E1 -38219.374,E2 -38219.374} C_VEL
LIN {X 0,Y 26.479,Z 636.255,A -85,B 0,C 180,E1 -38249.998,E2 -38249.998} C_VEL
LIN {X 0,Y 32.845,Z 633.98,A -85,B 0,C 180,E1 -38275.244,E2 -38275.244} C_VEL
LIN {X 0,Y 43.756,Z 630.396,A -85,B 0,C 180,E1 -38289.814,E2 -38289.814} C_VEL
LIN {X 0,Y 56.433,Z 625.316,A -85,B 0,C 180,E1 -38298.134,E2 -38298.134} C_VEL
LIN {X 0,Y 61.146,Z 623.069,A -85,B 0,C 180,E1 -38300.339,E2 -38300.339} C_VEL
LIN {X 0,Y 60.528,Z 622.259,A -85,B 0,C 180,E1 -38302.593,E2 -38302.593} C_VEL
LIN {X 0,Y 56.241,Z 620.759,A -85,B 0,C 180,E1 -38310.123,E2 -38310.123} C_VEL
LIN {X 0,Y 50.761,Z 618.673,A -85,B 0,C 180,E1 -38324.996,E2 -38324.996} C_VEL
LIN {X 0,Y 51.493,Z 614.884,A -85,B 0,C 180,E1 -38347.82,E2 -38347.82} C_VEL
LIN {X 0,Y 60.987,Z 610.124,A -85,B 0,C 180,E1 -38366.684,E2 -38366.684} C_VEL
LIN {X 0,Y 61.383,Z 609.964,A -85,B 0,C 180,E1 -38367.16,E2 -38367.16} C_VEL
LIN {X 0,Y 50.559,Z 616.822,A -85,B 0,C 180,E1 -38373.776,E2 -38373.776} C_VEL
LIN {X 0,Y 39.624,Z 622.739,A -85,B 0,C 180,E1 -38385.003,E2 -38385.003} C_VEL
LIN {X 0,Y 30.999,Z 627.103,A -85,B 0,C 180,E1 -38403.136,E2 -38403.136} C_VEL
LIN {X 0,Y 27.004,Z 630.064,A -85,B 0,C 180,E1 -38430.002,E2 -38430.002} C_VEL
LIN {X 0,Y 29.44,Z 631.72,A -85,B 0,C 180,E1 -38458.416,E2 -38458.416} C_VEL
LIN {X 0,Y 37.141,Z 632.092,A -85,B 0,C 180,E1 -38478.973,E2 -38478.973} C_VEL
LIN {X 0,Y 47.795,Z 631.153,A -85,B 0,C 180,E1 -38491.563,E2 -38491.563} C_VEL
LIN {X 0,Y 53.916,Z 630.144,A -85,B 0,C 180,E1 -38496.11,E2 -38496.11} C_VEL
LIN {X 0,Y 54.33,Z 630.105,A -85,B 0,C 180,E1 -38497.368,E2 -38497.368} C_VEL
LIN {X 0,Y 53.501,Z 630.339,A -85,B 0,C 180,E1 -38499.756,E2 -38499.756} C_VEL
LIN {X 0,Y 51.047,Z 630.92,A -85,B 0,C 180,E1 -38502.719,E2 -38502.719} C_VEL
LIN {X 0,Y 43.282,Z 632.682,A -85,B 0,C 180,E1 -38510.208,E2 -38510.208} C_VEL
LIN {X 0,Y 40.919,Z 633.296,A -85,B 0,C 180,E1 -38515.045,E2 -38515.045} C_VEL
LIN {X 0,Y 40.632,Z 633.408,A -85,B 0,C 180,E1 -38516.177,E2 -38516.177} C_VEL
LIN {X 0,Y 39.228,Z 635.273,A -85,B 0,C 180,E1 -38537.394,E2 -38537.394} C_VEL
LIN {X 0,Y 37.464,Z 635.686,A -85,B 0,C 180,E1 -38540.796,E2 -38540.796} C_VEL
LIN {X 0,Y 26.034,Z 636.516,A -85,B 0,C 180,E1 -38556.176,E2 -38556.176} C_VEL
LIN {X 0,Y 19.176,Z 636.097,A -85,B 0,C 180,E1 -38588.573,E2 -38588.573} C_VEL
LIN {X 0,Y 22.402,Z 634.297,A -85,B 0,C 180,E1 -38630.296,E2 -38630.296} C_VEL
LIN {X 0,Y 32.181,Z 631.479,A -85,B 0,C 180,E1 -38650.764,E2 -38650.764} C_VEL
LIN {X 0,Y 45.12,Z 627.145,A -85,B 0,C 180,E1 -38660.911,E2 -38660.911} C_VEL
LIN {X 0,Y 51.924,Z 624.392,A -85,B 0,C 180,E1 -38664.034,E2 -38664.034} C_VEL
LIN {X 0,Y 50.788,Z 623.921,A -85,B 0,C 180,E1 -38666.521,E2 -38666.521} C_VEL
LIN {X 0,Y 44.873,Z 621.994,A -85,B 0,C 180,E1 -38681.811,E2 -38681.811} C_VEL
LIN {X 0,Y 43.804,Z 619.613,A -85,B 0,C 180,E1 -38700.002,E2 -38700.002} C_VEL
LIN {X 0,Y 47.78,Z 616.817,A -85,B 0,C 180,E1 -38717.052,E2 -38717.052} C_VEL
LIN {X 0,Y 51.34,Z 615.303,A -85,B 0,C 180,E1 -38724.163,E2 -38724.163} C_VEL
LIN {X 0,Y 40.843,Z 620.889,A -85,B 0,C 180,E1 -38730.967,E2 -38730.967} C_VEL
LIN {X 0,Y 29.596,Z 625.963,A -85,B 0,C 180,E1 -38744.768,E2 -38744.768} C_VEL
LIN {X 0,Y 21.485,Z 629.585,A -85,B 0,C 180,E1 -38770.976,E2 -38770.976} C_VEL
LIN {X 0,Y 20.644,Z 631.859,A -85,B 0,C 180,E1 -38809.838,E2 -38809.838} C_VEL
LIN {X 0,Y 27.739,Z 632.843,A -85,B 0,C 180,E1 -38839.252,E2 -38839.252} C_VEL
LIN {X 0,Y 38.677,Z 632.545,A -85,B 0,C 180,E1 -38854.897,E2 -38854.897} C_VEL
LIN {X 0,Y 44.851,Z 631.888,A -85,B 0,C 180,E1 -38859.564,E2 -38859.564} C_VEL
LIN {X 0,Y 45.471,Z 631.913,A -85,B 0,C 180,E1 -38862.054,E2 -38862.054} C_VEL
LIN {X 0,Y 40.632,Z 633.408,A -85,B 0,C 180,E1 -38876.177,E2 -38876.177} C_VEL
LIN {X 0,Y 38.917,Z 633.955,A -85,B 0,C 180,E1 -38880.9,E2 -38880.9} C_VEL
LIN {X 0,Y 36.358,Z 634.529,A -85,B 0,C 180,E1 -38885.093,E2 -38885.093} C_VEL
LIN {X 0,Y 33.258,Z 635.026,A -85,B 0,C 180,E1 -38889.033,E2 -38889.033} C_VEL
LIN {X 0,Y 29.897,Z 635.395,A -85,B 0,C 180,E1 -38892.759,E2 -38892.759} C_VEL
LIN {X 0,Y 22.188,Z 635.749,A -85,B 0,C 180,E1 -38902.224,E2 -38902.224} C_VEL
LIN {X 0,Y 15.34,Z 635.541,A -85,B 0,C 180,E1 -38919.606,E2 -38919.606} C_VEL
LIN {X 0,Y 12.125,Z 634.594,A -85,B 0,C 180,E1 -38969.995,E2 -38969.995} C_VEL
LIN {X 0,Y 20.751,Z 632.255,A -85,B 0,C 180,E1 -39012.459,E2 -39012.459} C_VEL
LIN {X 0,Y 33.924,Z 628.597,A -85,B 0,C 180,E1 -39025.677,E2 -39025.677} C_VEL
LIN {X 0,Y 40.937,Z 626.228,A -85,B 0,C 180,E1 -39028.815,E2 -39028.815} C_VEL
LIN {X 0,Y 41.618,Z 625.843,A -85,B 0,C 180,E1 -39029.677,E2 -39029.677} C_VEL
LIN {X 0,Y 37.257,Z 623.805,A -85,B 0,C 180,E1 -39049.166,E2 -39049.166} C_VEL
LIN {X 0,Y 40.755,Z 620.32,A -85,B 0,C 180,E1 -39077.492,E2 -39077.492} C_VEL
LIN {X 0,Y 40.505,Z 620.486,A -85,B 0,C 180,E1 -39080.237,E2 -39080.237} C_VEL
LIN {X 0,Y 28.171,Z 625.718,A -85,B 0,C 180,E1 -39089.518,E2 -39089.518} C_VEL
LIN {X 0,Y 19.487,Z 628.797,A -85,B 0,C 180,E1 -39104.044,E2 -39104.044} C_VEL
LIN {X 0,Y 12.858,Z 631.703,A -85,B 0,C 180,E1 -39150.005,E2 -39150.005} C_VEL
LIN {X 0,Y 18.267,Z 633.304,A -85,B 0,C 180,E1 -39200.081,E2 -39200.081} C_VEL
LIN {X 0,Y 29.805,Z 633.623,A -85,B 0,C 180,E1 -39220.062,E2 -39220.062} C_VEL
LIN {X 0,Y 34.085,Z 633.433,A -85,B 0,C 180,E1 -39223.631,E2 -39223.631} C_VEL
LIN {X 0,Y 35.562,Z 633.434,A -85,B 0,C 180,E1 -39226.493,E2 -39226.493} C_VEL
LIN {X 0,Y 31.992,Z 635.087,A -85,B 0,C 180,E1 -39249.448,E2 -39249.448} C_VEL
LIN {X 0,Y 29.644,Z 635.451,A -85,B 0,C 180,E1 -39253.664,E2 -39253.664} C_VEL
LIN {X 0,Y 16.853,Z 635.659,A -85,B 0,C 180,E1 -39273.765,E2 -39273.765} C_VEL
LIN {X 0,Y 15.34,Z 635.541,A -85,B 0,C 180,E1 -39279.606,E2 -39279.606} C_VEL
LIN {X 0,Y 11.85,Z 635.13,A -85,B 0,C 180,E1 -39299.867,E2 -39299.867} C_VEL
LIN {X 0,Y 10.138,Z 633.684,A -85,B 0,C 180,E1 -39352.145,E2 -39352.145} C_VEL
LIN {X 0,Y 16.046,Z 631.611,A -85,B 0,C 180,E1 -39387.127,E2 -39387.127} C_VEL
LIN {X 0,Y 21.37,Z 630.16,A -85,B 0,C 180,E1 -39393.737,E2 -39393.737} C_VEL
LIN {X 0,Y 30.45,Z 627.703,A -85,B 0,C 180,E1 -39396.94,E2 -39396.94} C_VEL
LIN {X 0,Y 30.759,Z 626.418,A -85,B 0,C 180,E1 -39406.841,E2 -39406.841} C_VEL
LIN {X 0,Y 31.925,Z 624.255,A -85,B 0,C 180,E1 -39430.893,E2 -39430.893} C_VEL
LIN {X 0,Y 30.418,Z 624.806,A -85,B 0,C 180,E1 -39433.129,E2 -39433.129} C_VEL
LIN {X 0,Y 22.065,Z 627.686,A -85,B 0,C 180,E1 -39437.768,E2 -39437.768} C_VEL
LIN {X 0,Y 9.351,Z 631.248,A -85,B 0,C 180,E1 -39461.5,E2 -39461.5} C_VEL
LIN {X 0,Y 8.76,Z 633.47,A -85,B 0,C 180,E1 -39563.108,E2 -39563.108} C_VEL
LIN {X 0,Y 21.373,Z 634.402,A -85,B 0,C 180,E1 -39589.494,E2 -39589.494} C_VEL
LIN {X 0,Y 23.501,Z 634.457,A -85,B 0,C 180,E1 -39591.095,E2 -39591.095} C_VEL
LIN {X 0,Y 25.877,Z 634.583,A -85,B 0,C 180,E1 -39595.967,E2 -39595.967} C_VEL
LIN {X 0,Y 25.422,Z 634.789,A -85,B 0,C 180,E1 -39599.996,E2 -39599.996} C_VEL
LIN {X 0,Y 21.042,Z 634.947,A -85,B 0,C 180,E1 -39602.932,E2 -39602.932} C_VEL
LIN {X 0,Y 7.849,Z 634.47,A -85,B 0,C 180,E1 -39626.799,E2 -39626.799} C_VEL
LIN {X 0,Y 9.561,Z 632.744,A -85,B 0,C 180,E1 -39737.095,E2 -39737.095} C_VEL
LIN {X 0,Y 21.37,Z 630.16,A -85,B 0,C 180,E1 -39753.737,E2 -39753.737} C_VEL
LIN {X 0,Y 22.421,Z 629.707,A -85,B 0,C 180,E1 -39756.773,E2 -39756.773} C_VEL
LIN {X 0,Y 22.711,Z 629.124,A -85,B 0,C 180,E1 -39762.824,E2 -39762.824} C_VEL
LIN {X 0,Y 23.255,Z 628.15,A -85,B 0,C 180,E1 -39774.375,E2 -39774.375} C_VEL
LIN {X 0,Y 23.596,Z 627.971,A -85,B 0,C 180,E1 -39775.719,E2 -39775.719} C_VEL
LIN {X 0,Y 23.784,Z 627.882,A -85,B 0,C 180,E1 -39776.314,E2 -39776.314} C_VEL
LIN {X 0,Y 21.015,Z 628.545,A -85,B 0,C 180,E1 -39779.143,E2 -39779.143} C_VEL
LIN {X 0,Y 14.02,Z 630.489,A -85,B 0,C 180,E1 -39777.652,E2 -39777.652} C_VEL
LIN {X 0,Y 14.04,Z 630.534,A -85,B 0,C 180,E1 -39776.135,E2 -39776.135} C_VEL
LIN {X 0,Y 22.584,Z 628.476,A -85,B 0,C 180,E1 -39772.174,E2 -39772.174} C_VEL
LIN {X 0,Y 23.596,Z 627.971,A -85,B 0,C 180,E1 -39775.719,E2 -39775.719} C_VEL
LIN {X 0,Y 23.596,Z 627.971,A -85,B 0,C 180,E1 -39775.719,E2 -39775.719}

QRS_NEXT_CUT()

QRS_NEXT()
QRS_HOME()

END
